Universal Robots PolyScope program: functionTest.urp

Program functionTest (installation=default directory=/home/ur/ursim/ursim-5.11.0.108249/programs createdIn=5.11.0.108249 lastSavedIn=5.11.0.108249 robotSerialNumber=20205500065)
Calibrated DH parameters: a=[0, -0.425, -0.3922, 0, 0, 0]; d=[0.1625, 0, 0, 0.1333, 0.0997, 0.0996]; alpha=[1.570796, 0, 0, 1.570796, -1.570796, 0]; deltaTheta=[0, 0, 0, 0, 0, 0]
BeforeStart
  var_1 := 0
Robot Program (runOnlyOnce=false)
  var_1 := ci_add(var_1,1)
  Wait Sleep waitTime=0.3
